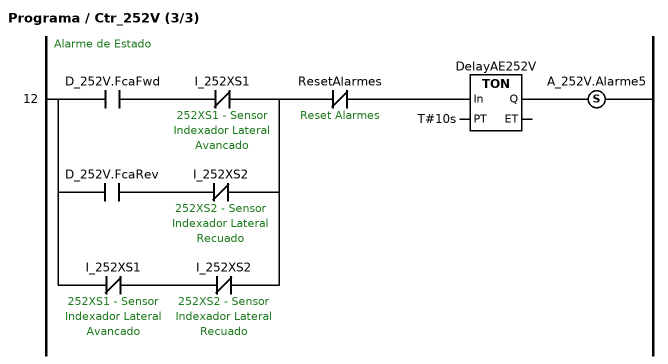
(* [picture p96: Programa / Ctr_252V, rungs 12-12] *)
(* Rung 12: Alarme de Estado *)
DelayAE252V(In := ((D_252V.FcaFwd AND NOT I_252XS1) OR (D_252V.FcaRev AND NOT I_252XS2) OR (NOT I_252XS1 AND NOT I_252XS2)) AND NOT ResetAlarmes, PT := T#10s);
IF DelayAE252V.Q THEN A_252V.Alarme5 := TRUE; END_IF;

(* Section Ctr_310M1: ladder, written here as Structured Text *)

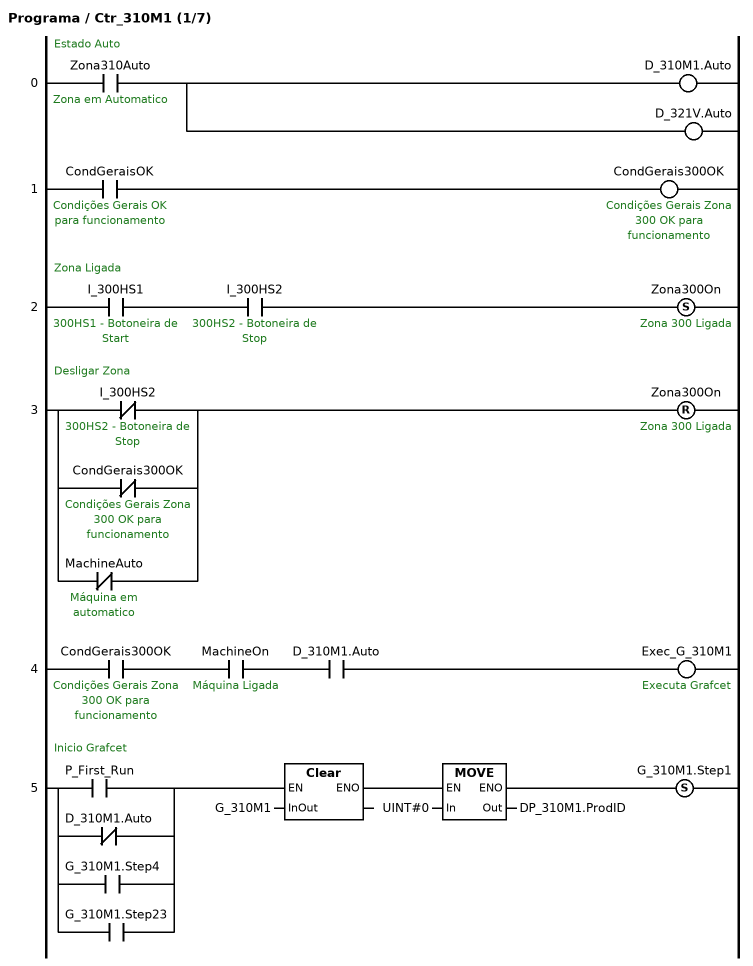
(* Rung 0: Estado Auto *)
D_310M1.Auto := Zona310Auto;
D_321V.Auto := Zona310Auto;
(* Rung 1 *)
CondGerais300OK := CondGeraisOK;
(* Rung 2: Zona Ligada *)
IF I_300HS1 AND I_300HS2 THEN Zona300On := TRUE; END_IF;
(* Rung 3: Desligar Zona *)
IF NOT I_300HS2 OR NOT CondGerais300OK OR NOT MachineAuto THEN Zona300On := FALSE; END_IF;
(* Rung 4 *)
Exec_G_310M1 := CondGerais300OK AND MachineOn AND D_310M1.Auto;
(* Rung 5: Inicio Grafcet *)
_p186 := P_First_Run OR NOT D_310M1.Auto OR G_310M1.Step4 OR G_310M1.Step23;
IF _p186 THEN
    Clear(InOut := G_310M1);
    DP_310M1.ProdID := UINT#0;
    G_310M1.Step1 := TRUE;
END_IF;

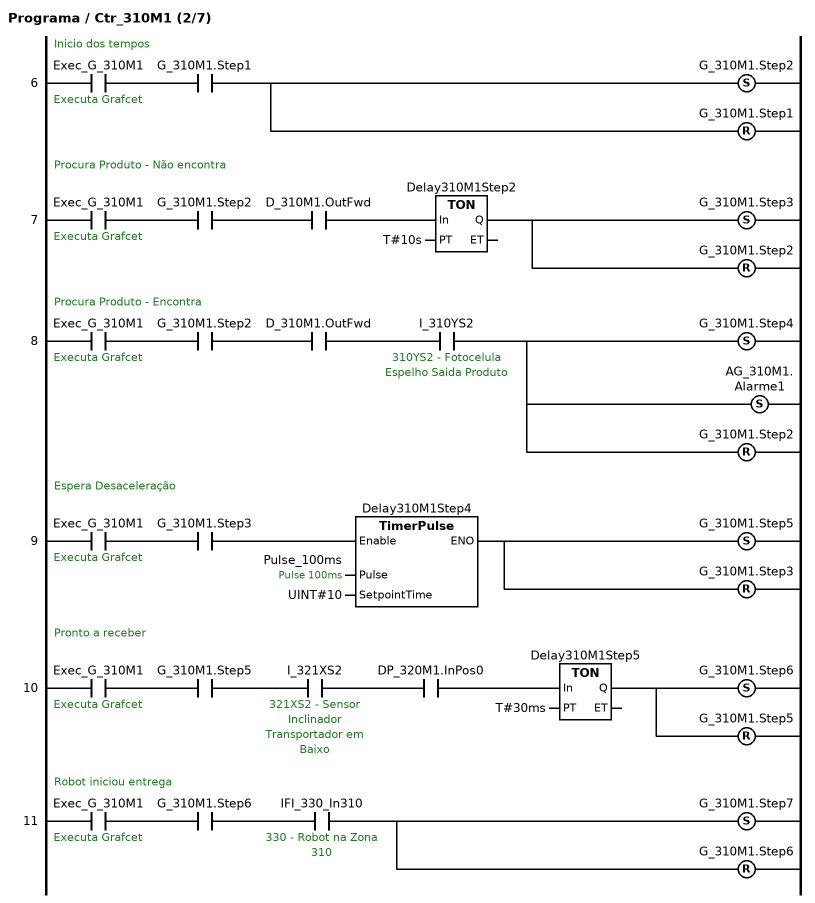
(* Rung 6: Inicio dos tempos *)
_p187 := Exec_G_310M1 AND G_310M1.Step1;
IF _p187 THEN
    G_310M1.Step2 := TRUE;
    G_310M1.Step1 := FALSE;
END_IF;
(* Rung 7: Procura Produto - Não encontra *)
Delay310M1Step2(In := Exec_G_310M1 AND G_310M1.Step2 AND D_310M1.OutFwd, PT := T#10s);
IF Delay310M1Step2.Q THEN
    G_310M1.Step3 := TRUE;
    G_310M1.Step2 := FALSE;
END_IF;
(* Rung 8: Procura Produto - Encontra *)
_p188 := Exec_G_310M1 AND G_310M1.Step2 AND D_310M1.OutFwd AND I_310YS2;
IF _p188 THEN
    G_310M1.Step4 := TRUE;
    AG_310M1.Alarme1 := TRUE;
    G_310M1.Step2 := FALSE;
END_IF;
(* Rung 9: Espera Desaceleração *)
Delay310M1Step4(Enable := Exec_G_310M1 AND G_310M1.Step3, Pulse := Pulse_100ms, SetpointTime := UINT#10);
IF Delay310M1Step4.ENO THEN
    G_310M1.Step5 := TRUE;
    G_310M1.Step3 := FALSE;
END_IF;
(* Rung 10: Pronto a receber *)
Delay310M1Step5(In := Exec_G_310M1 AND G_310M1.Step5 AND I_321XS2 AND DP_320M1.InPos0, PT := T#30ms);
IF Delay310M1Step5.Q THEN
    G_310M1.Step6 := TRUE;
    G_310M1.Step5 := FALSE;
END_IF;
(* Rung 11: Robot iniciou entrega *)
_p189 := Exec_G_310M1 AND G_310M1.Step6 AND IFI_330_In310;
IF _p189 THEN
    G_310M1.Step7 := TRUE;
    G_310M1.Step6 := FALSE;
END_IF;

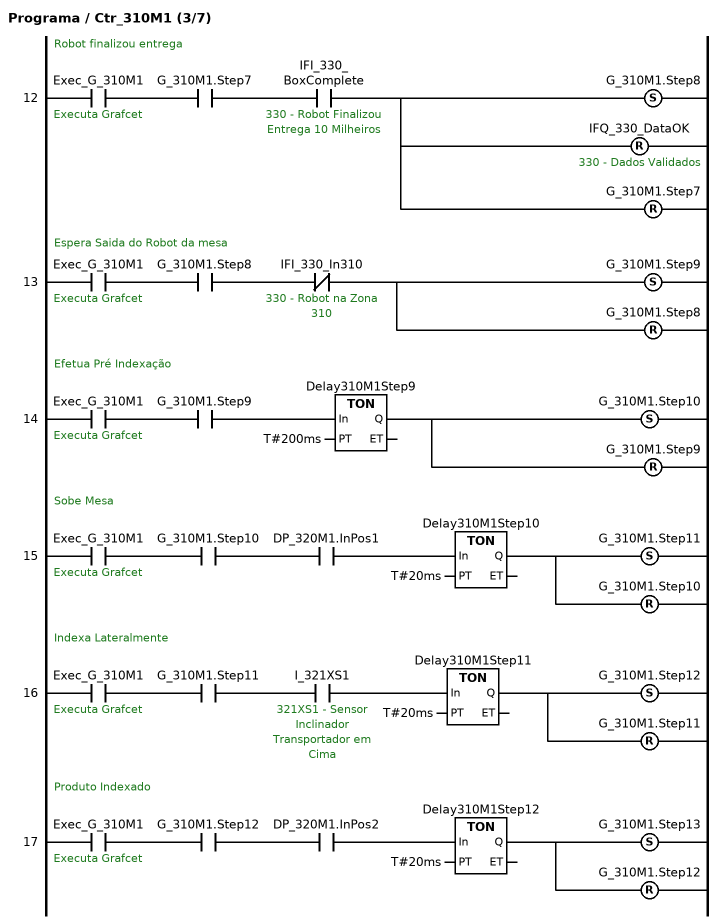
(* Rung 12: Robot finalizou entrega *)
_p190 := Exec_G_310M1 AND G_310M1.Step7 AND IFI_330_BoxComplete;
IF _p190 THEN
    G_310M1.Step8 := TRUE;
    IFQ_330_DataOK := FALSE;
    G_310M1.Step7 := FALSE;
END_IF;
(* Rung 13: Espera Saida do Robot da mesa *)
_p191 := Exec_G_310M1 AND G_310M1.Step8 AND NOT IFI_330_In310;
IF _p191 THEN
    G_310M1.Step9 := TRUE;
    G_310M1.Step8 := FALSE;
END_IF;
(* Rung 14: Efetua Pré Indexação *)
Delay310M1Step9(In := Exec_G_310M1 AND G_310M1.Step9, PT := T#200ms);
IF Delay310M1Step9.Q THEN
    G_310M1.Step10 := TRUE;
    G_310M1.Step9 := FALSE;
END_IF;
(* Rung 15: Sobe Mesa *)
Delay310M1Step10(In := Exec_G_310M1 AND G_310M1.Step10 AND DP_320M1.InPos1, PT := T#20ms);
IF Delay310M1Step10.Q THEN
    G_310M1.Step11 := TRUE;
    G_310M1.Step10 := FALSE;
END_IF;
(* Rung 16: Indexa Lateralmente *)
Delay310M1Step11(In := Exec_G_310M1 AND G_310M1.Step11 AND I_321XS1, PT := T#20ms);
IF Delay310M1Step11.Q THEN
    G_310M1.Step12 := TRUE;
    G_310M1.Step11 := FALSE;
END_IF;
(* Rung 17: Produto Indexado *)
Delay310M1Step12(In := Exec_G_310M1 AND G_310M1.Step12 AND DP_320M1.InPos2, PT := T#20ms);
IF Delay310M1Step12.Q THEN
    G_310M1.Step13 := TRUE;
    G_310M1.Step12 := FALSE;
END_IF;

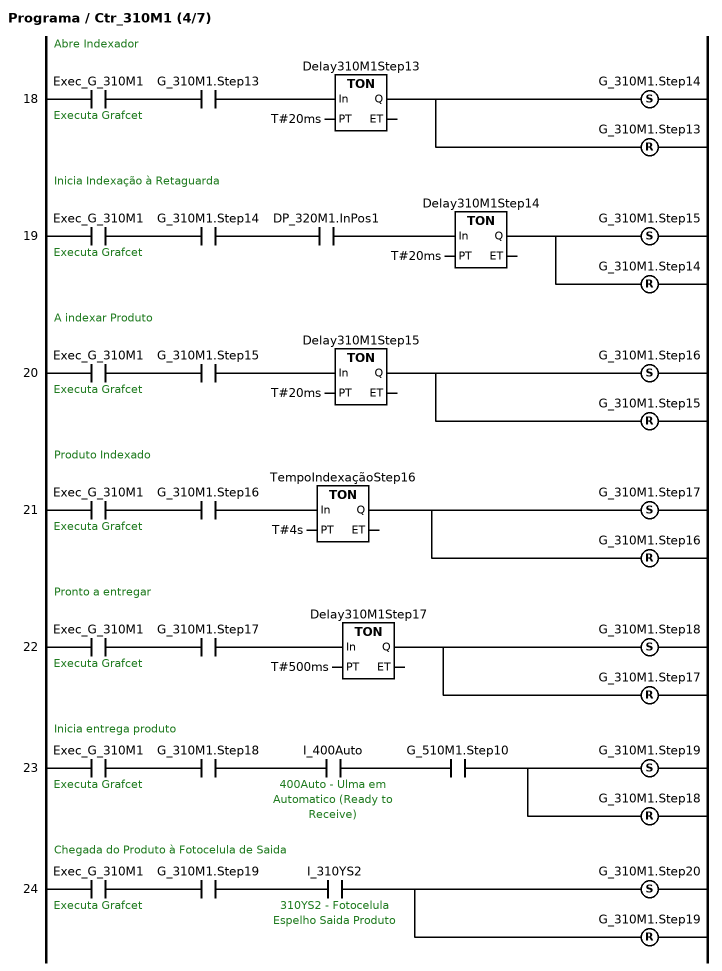
(* Rung 18: Abre Indexador *)
Delay310M1Step13(In := Exec_G_310M1 AND G_310M1.Step13, PT := T#20ms);
IF Delay310M1Step13.Q THEN
    G_310M1.Step14 := TRUE;
    G_310M1.Step13 := FALSE;
END_IF;
(* Rung 19: Inicia Indexação à Retaguarda *)
Delay310M1Step14(In := Exec_G_310M1 AND G_310M1.Step14 AND DP_320M1.InPos1, PT := T#20ms);
IF Delay310M1Step14.Q THEN
    G_310M1.Step15 := TRUE;
    G_310M1.Step14 := FALSE;
END_IF;
(* Rung 20: A indexar Produto *)
Delay310M1Step15(In := Exec_G_310M1 AND G_310M1.Step15, PT := T#20ms);
IF Delay310M1Step15.Q THEN
    G_310M1.Step16 := TRUE;
    G_310M1.Step15 := FALSE;
END_IF;
(* Rung 21: Produto Indexado *)
TempoIndexaçãoStep16(In := Exec_G_310M1 AND G_310M1.Step16, PT := T#4s);
IF TempoIndexaçãoStep16.Q THEN
    G_310M1.Step17 := TRUE;
    G_310M1.Step16 := FALSE;
END_IF;
(* Rung 22: Pronto a entregar *)
Delay310M1Step17(In := Exec_G_310M1 AND G_310M1.Step17, PT := T#500ms);
IF Delay310M1Step17.Q THEN
    G_310M1.Step18 := TRUE;
    G_310M1.Step17 := FALSE;
END_IF;
(* Rung 23: Inicia entrega produto *)
_p192 := Exec_G_310M1 AND G_310M1.Step18 AND I_400Auto AND G_510M1.Step10;
IF _p192 THEN
    G_310M1.Step19 := TRUE;
    G_310M1.Step18 := FALSE;
END_IF;
(* Rung 24: Chegada do Produto à Fotocelula de Saida *)
_p193 := Exec_G_310M1 AND G_310M1.Step19 AND I_310YS2;
IF _p193 THEN
    G_310M1.Step20 := TRUE;
    G_310M1.Step19 := FALSE;
END_IF;

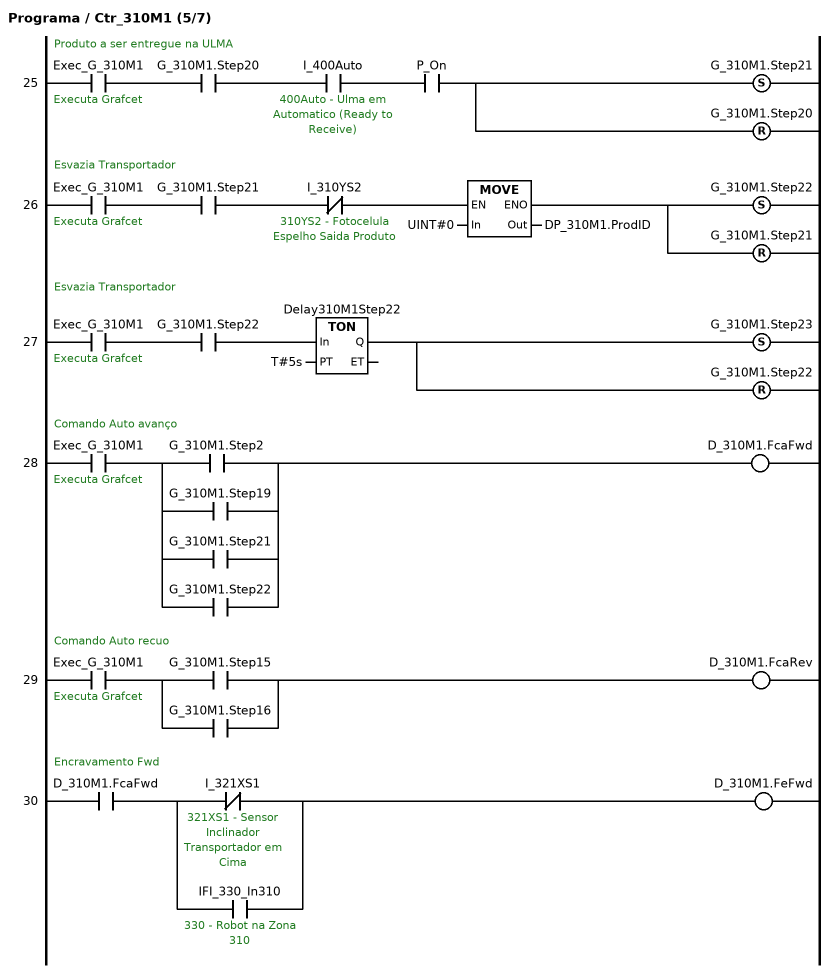
(* Rung 25: Produto a ser entregue na ULMA *)
_p194 := Exec_G_310M1 AND G_310M1.Step20 AND I_400Auto AND P_On;
IF _p194 THEN
    G_310M1.Step21 := TRUE;
    G_310M1.Step20 := FALSE;
END_IF;
(* Rung 26: Esvazia Transportador *)
IF Exec_G_310M1 AND G_310M1.Step21 AND NOT I_310YS2 THEN DP_310M1.ProdID := UINT#0; END_IF;
_p195 := Exec_G_310M1 AND G_310M1.Step21 AND NOT I_310YS2;
IF _p195 THEN
    G_310M1.Step22 := TRUE;
    G_310M1.Step21 := FALSE;
END_IF;
(* Rung 27: Esvazia Transportador *)
Delay310M1Step22(In := Exec_G_310M1 AND G_310M1.Step22, PT := T#5s);
IF Delay310M1Step22.Q THEN
    G_310M1.Step23 := TRUE;
    G_310M1.Step22 := FALSE;
END_IF;
(* Rung 28: Comando Auto avanço *)
D_310M1.FcaFwd := Exec_G_310M1 AND (G_310M1.Step2 OR G_310M1.Step19 OR G_310M1.Step21 OR G_310M1.Step22);
(* Rung 29: Comando Auto recuo *)
D_310M1.FcaRev := Exec_G_310M1 AND (G_310M1.Step15 OR G_310M1.Step16);
(* Rung 30: Encravamento Fwd *)
D_310M1.FeFwd := D_310M1.FcaFwd AND (NOT I_321XS1 OR IFI_330_In310);

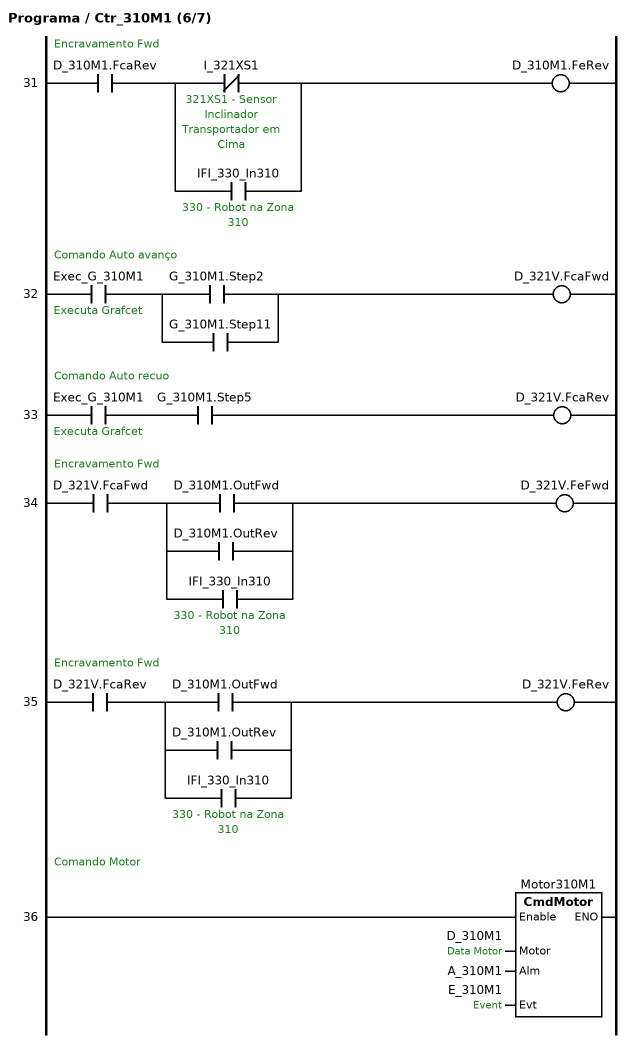
(* Rung 31: Encravamento Fwd *)
D_310M1.FeRev := D_310M1.FcaRev AND (NOT I_321XS1 OR IFI_330_In310);
(* Rung 32: Comando Auto avanço *)
D_321V.FcaFwd := Exec_G_310M1 AND (G_310M1.Step2 OR G_310M1.Step11);
(* Rung 33: Comando Auto recuo *)
D_321V.FcaRev := Exec_G_310M1 AND G_310M1.Step5;
(* Rung 34: Encravamento Fwd *)
D_321V.FeFwd := D_321V.FcaFwd AND (D_310M1.OutFwd OR D_310M1.OutRev OR IFI_330_In310);
(* Rung 35: Encravamento Fwd *)
D_321V.FeRev := D_321V.FcaRev AND (D_310M1.OutFwd OR D_310M1.OutRev OR IFI_330_In310);
(* Rung 36: Comando Motor *)
Motor310M1(Enable := TRUE, Motor := D_310M1, Alm := A_310M1, Evt := E_310M1);

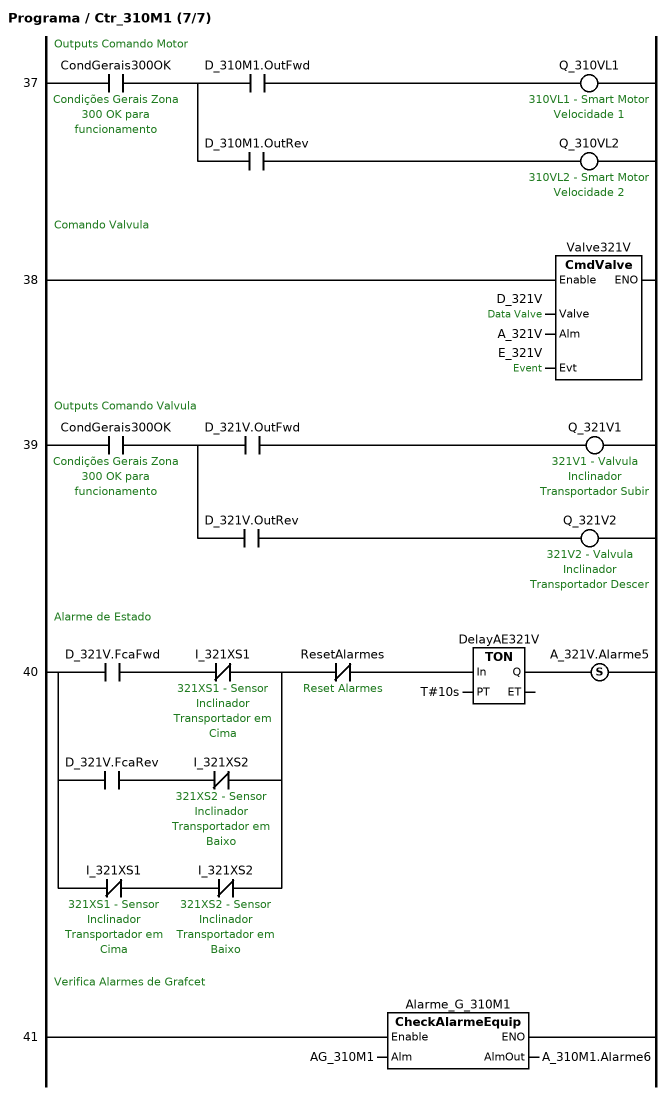
(* Rung 37: Outputs Comando Motor *)
Q_310VL1 := CondGerais300OK AND D_310M1.OutFwd;
Q_310VL2 := CondGerais300OK AND D_310M1.OutRev;
(* Rung 38: Comando Valvula *)
Valve321V(Enable := TRUE, Valve := D_321V, Alm := A_321V, Evt := E_321V);
(* Rung 39: Outputs Comando Valvula *)
Q_321V1 := CondGerais300OK AND D_321V.OutFwd;
Q_321V2 := CondGerais300OK AND D_321V.OutRev;
(* Rung 40: Alarme de Estado *)
DelayAE321V(In := ((D_321V.FcaFwd AND NOT I_321XS1) OR (D_321V.FcaRev AND NOT I_321XS2) OR (NOT I_321XS1 AND NOT I_321XS2)) AND NOT ResetAlarmes, PT := T#10s);
IF DelayAE321V.Q THEN A_321V.Alarme5 := TRUE; END_IF;
(* Rung 41: Verifica Alarmes de Grafcet *)
Alarme_G_310M1(Enable := TRUE, Alm := AG_310M1, AlmOut => A_310M1.Alarme6);

(* Section Ctr_320M1_Servo: ladder, written here as Structured Text *)

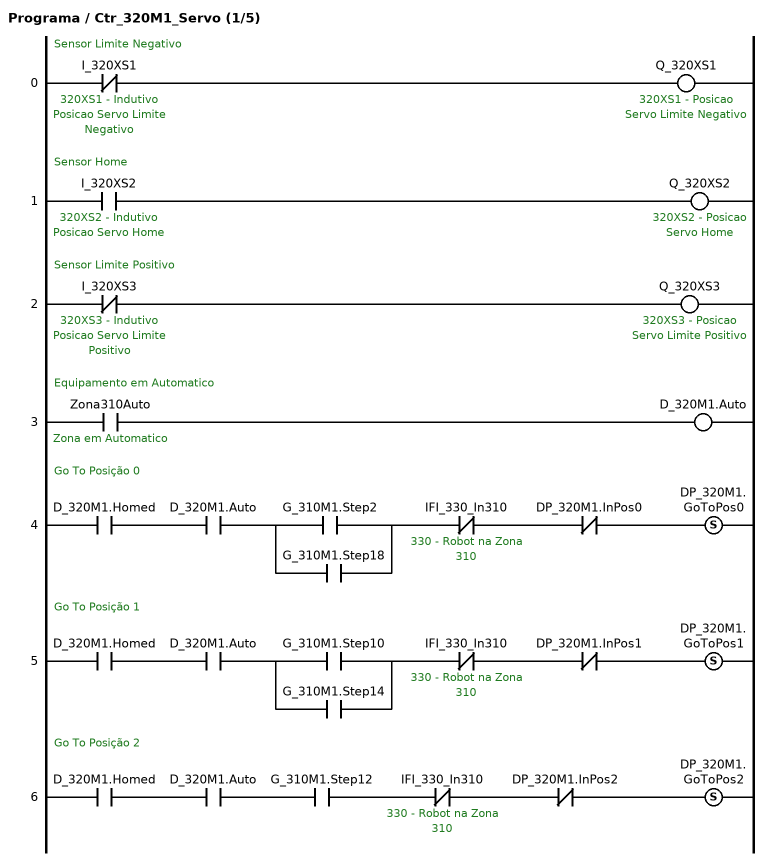
(* Rung 0: Sensor Limite Negativo *)
Q_320XS1 := NOT I_320XS1;
(* Rung 1: Sensor Home *)
Q_320XS2 := I_320XS2;
(* Rung 2: Sensor Limite Positivo *)
Q_320XS3 := NOT I_320XS3;
(* Rung 3: Equipamento em Automatico *)
D_320M1.Auto := Zona310Auto;
(* Rung 4: Go To Posição 0 *)
IF D_320M1.Homed AND D_320M1.Auto AND (G_310M1.Step2 OR G_310M1.Step18) AND NOT IFI_330_In310 AND NOT DP_320M1.InPos0 THEN
    DP_320M1.GoToPos0 := TRUE;
END_IF;
(* Rung 5: Go To Posição 1 *)
IF D_320M1.Homed AND D_320M1.Auto AND (G_310M1.Step10 OR G_310M1.Step14) AND NOT IFI_330_In310 AND NOT DP_320M1.InPos1 THEN
    DP_320M1.GoToPos1 := TRUE;
END_IF;
(* Rung 6: Go To Posição 2 *)
IF D_320M1.Homed AND D_320M1.Auto AND G_310M1.Step12 AND NOT IFI_330_In310 AND NOT DP_320M1.InPos2 THEN
    DP_320M1.GoToPos2 := TRUE;
END_IF;

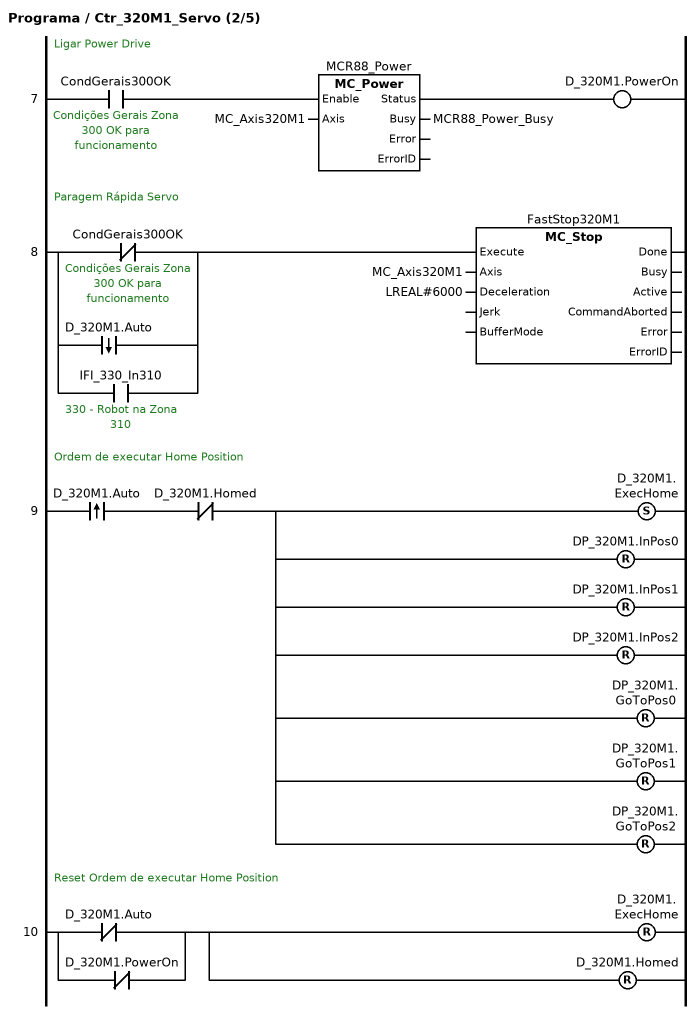
(* Rung 7: Ligar Power Drive *)
MCR88_Power(Enable := CondGerais300OK, Axis := MC_Axis320M1, Busy => MCR88_Power_Busy);
D_320M1.PowerOn := MCR88_Power.Status;
(* Rung 8: Paragem Rápida Servo *)
_e196(CLK := D_320M1.Auto);
FastStop320M1(Execute := NOT CondGerais300OK OR _e196.Q OR IFI_330_In310, Axis := MC_Axis320M1, Deceleration := LREAL#6000);
(* Rung 9: Ordem de executar Home Position *)
_e197(CLK := D_320M1.Auto);
_p198 := _e197.Q AND NOT D_320M1.Homed;
IF _p198 THEN
    D_320M1.ExecHome := TRUE;
    DP_320M1.InPos0 := FALSE;
    DP_320M1.InPos1 := FALSE;
    DP_320M1.InPos2 := FALSE;
    DP_320M1.GoToPos0 := FALSE;
    DP_320M1.GoToPos1 := FALSE;
    DP_320M1.GoToPos2 := FALSE;
END_IF;
(* Rung 10: Reset Ordem de executar Home Position *)
_p199 := NOT D_320M1.Auto OR NOT D_320M1.PowerOn;
IF _p199 THEN
    D_320M1.ExecHome := FALSE;
    D_320M1.Homed := FALSE;
END_IF;

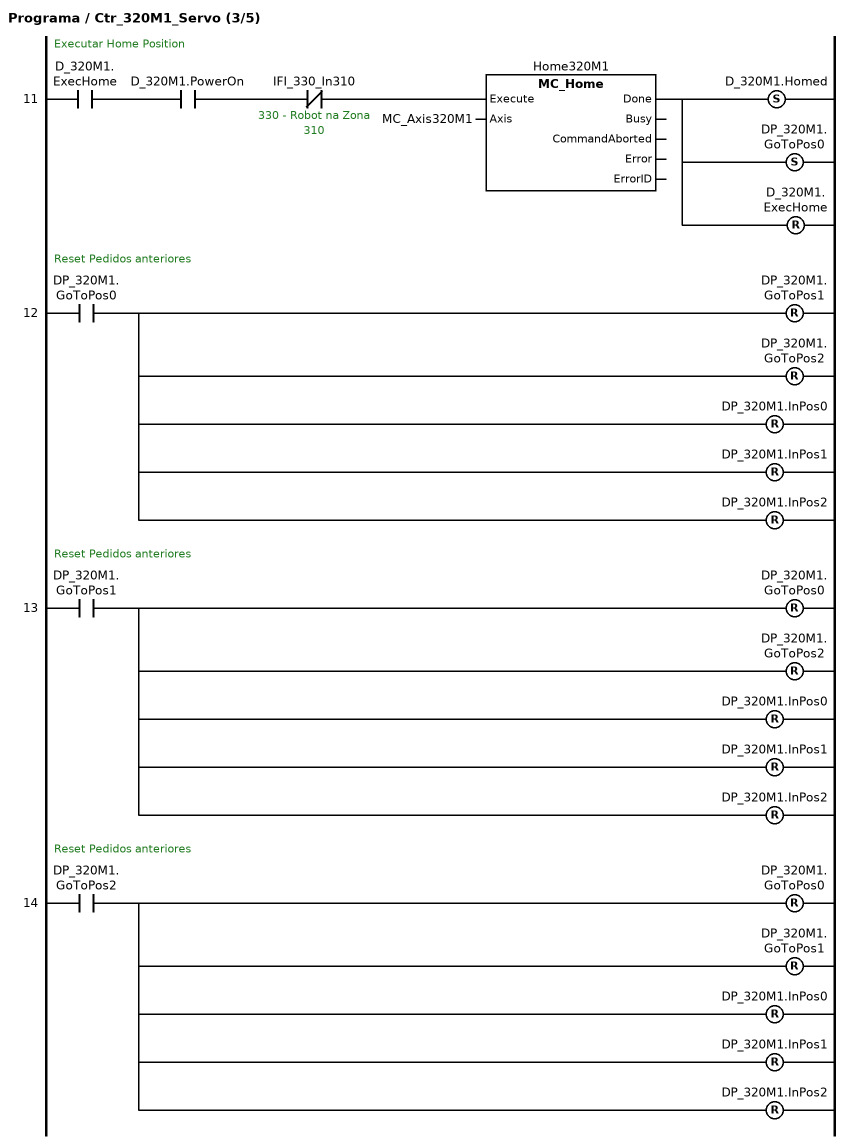
(* Rung 11: Executar Home Position *)
Home320M1(Execute := D_320M1.ExecHome AND D_320M1.PowerOn AND NOT IFI_330_In310, Axis := MC_Axis320M1);
IF Home320M1.Done THEN
    D_320M1.Homed := TRUE;
    DP_320M1.GoToPos0 := TRUE;
    D_320M1.ExecHome := FALSE;
END_IF;
(* Rung 12: Reset Pedidos anteriores *)
_p200 := DP_320M1.GoToPos0;
IF _p200 THEN
    DP_320M1.GoToPos1 := FALSE;
    DP_320M1.GoToPos2 := FALSE;
    DP_320M1.InPos0 := FALSE;
    DP_320M1.InPos1 := FALSE;
    DP_320M1.InPos2 := FALSE;
END_IF;
(* Rung 13: Reset Pedidos anteriores *)
_p201 := DP_320M1.GoToPos1;
IF _p201 THEN
    DP_320M1.GoToPos0 := FALSE;
    DP_320M1.GoToPos2 := FALSE;
    DP_320M1.InPos0 := FALSE;
    DP_320M1.InPos1 := FALSE;
    DP_320M1.InPos2 := FALSE;
END_IF;
(* Rung 14: Reset Pedidos anteriores *)
_p202 := DP_320M1.GoToPos2;
IF _p202 THEN
    DP_320M1.GoToPos0 := FALSE;
    DP_320M1.GoToPos1 := FALSE;
    DP_320M1.InPos0 := FALSE;
    DP_320M1.InPos1 := FALSE;
    DP_320M1.InPos2 := FALSE;
END_IF;

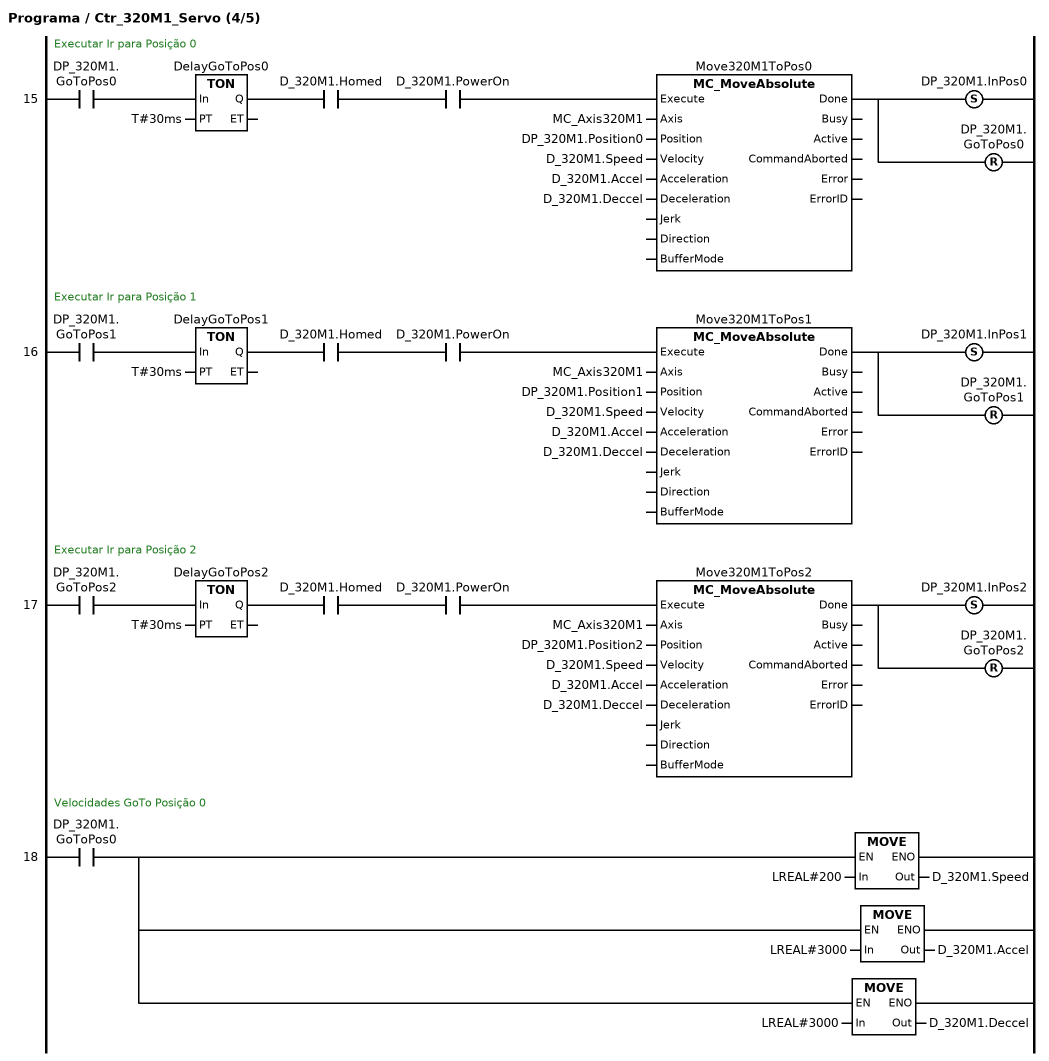
(* Rung 15: Executar Ir para Posição 0 *)
DelayGoToPos0(In := DP_320M1.GoToPos0, PT := T#30ms);
Move320M1ToPos0(Execute := DelayGoToPos0.Q AND D_320M1.Homed AND D_320M1.PowerOn, Axis := MC_Axis320M1, Position := DP_320M1.Position0, Velocity := D_320M1.Speed, Acceleration := D_320M1.Accel, Deceleration := D_320M1.Deccel);
IF Move320M1ToPos0.Done THEN
    DP_320M1.InPos0 := TRUE;
    DP_320M1.GoToPos0 := FALSE;
END_IF;
(* Rung 16: Executar Ir para Posição 1 *)
DelayGoToPos1(In := DP_320M1.GoToPos1, PT := T#30ms);
Move320M1ToPos1(Execute := DelayGoToPos1.Q AND D_320M1.Homed AND D_320M1.PowerOn, Axis := MC_Axis320M1, Position := DP_320M1.Position1, Velocity := D_320M1.Speed, Acceleration := D_320M1.Accel, Deceleration := D_320M1.Deccel);
IF Move320M1ToPos1.Done THEN
    DP_320M1.InPos1 := TRUE;
    DP_320M1.GoToPos1 := FALSE;
END_IF;
(* Rung 17: Executar Ir para Posição 2 *)
DelayGoToPos2(In := DP_320M1.GoToPos2, PT := T#30ms);
Move320M1ToPos2(Execute := DelayGoToPos2.Q AND D_320M1.Homed AND D_320M1.PowerOn, Axis := MC_Axis320M1, Position := DP_320M1.Position2, Velocity := D_320M1.Speed, Acceleration := D_320M1.Accel, Deceleration := D_320M1.Deccel);
IF Move320M1ToPos2.Done THEN
    DP_320M1.InPos2 := TRUE;
    DP_320M1.GoToPos2 := FALSE;
END_IF;
(* Rung 18: Velocidades GoTo Posição 0 *)
IF DP_320M1.GoToPos0 THEN
    D_320M1.Speed := LREAL#200;
    D_320M1.Accel := LREAL#3000;
    D_320M1.Deccel := LREAL#3000;
END_IF;

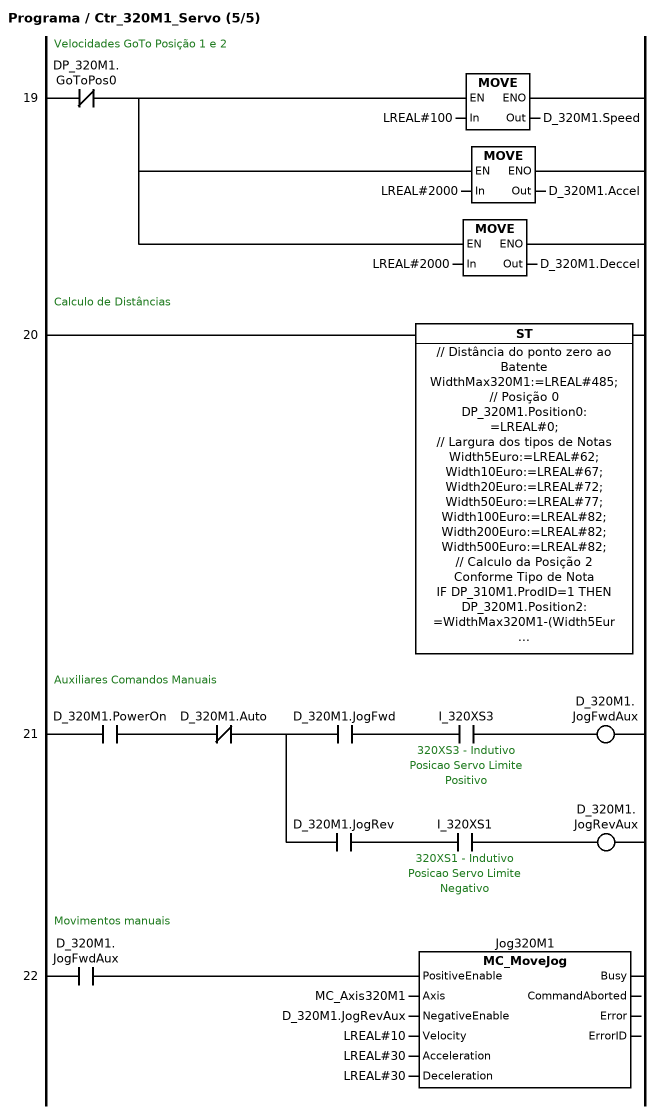
(* Rung 19: Velocidades GoTo Posição 1 e 2 *)
IF NOT DP_320M1.GoToPos0 THEN
    D_320M1.Speed := LREAL#100;
    D_320M1.Accel := LREAL#2000;
    D_320M1.Deccel := LREAL#2000;
END_IF;
(* Rung 20: Calculo de Distâncias *)
// Distância do ponto zero ao Batente

WidthMax320M1:=LREAL#485;

// Posição 0

DP_320M1.Position0:=LREAL#0;

// Largura dos tipos de Notas

Width5Euro:=LREAL#62;
Width10Euro:=LREAL#67;
Width20Euro:=LREAL#72;
Width50Euro:=LREAL#77;
Width100Euro:=LREAL#82;
Width200Euro:=LREAL#82;
Width500Euro:=LREAL#82;

// Calculo da Posição 2 Conforme Tipo de Nota

IF DP_310M1.ProdID=1 THEN DP_320M1.Position2:=WidthMax320M1-(Width5Euro*5); END_IF;
IF DP_310M1.ProdID=2 THEN DP_320M1.Position2:=WidthMax320M1-(Width10Euro*5); END_IF;
IF DP_310M1.ProdID=3 THEN DP_320M1.Position2:=WidthMax320M1-(Width20Euro*5); END_IF;	
IF DP_310M1.ProdID=4 THEN DP_320M1.Position2:=WidthMax320M1-(Width50Euro*5); END_IF;	
IF DP_310M1.ProdID=5 THEN DP_320M1.Position2:=WidthMax320M1-(Width100Euro*5); END_IF;
IF DP_310M1.ProdID=6 THEN DP_320M1.Position2:=WidthMax320M1-(Width200Euro*5); END_IF;
IF DP_310M1.ProdID=7 THEN DP_320M1.Position2:=WidthMax320M1-(Width500Euro*5); END_IF;
IF DP_310M1.ProdID<1 OR DP_310M1.ProdID>7 THEN DP_320M1.Position2:=WidthMax320M1-(Width500Euro*5); END_IF;
	
// Calculo da Posição 1 relativa a Posição 2

DP_320M1.Position1:=DP_320M1.Position2-LREAL#20;
(* Rung 21: Auxiliares Comandos Manuais *)
_p203 := D_320M1.PowerOn AND NOT D_320M1.Auto;
D_320M1.JogFwdAux := D_320M1.PowerOn AND NOT D_320M1.Auto AND D_320M1.JogFwd AND I_320XS3;
D_320M1.JogRevAux := _p203 AND D_320M1.JogRev AND I_320XS1;
(* Rung 22: Movimentos manuais *)
Jog320M1(PositiveEnable := D_320M1.JogFwdAux, Axis := MC_Axis320M1, NegativeEnable := D_320M1.JogRevAux, Velocity := LREAL#10, Acceleration := LREAL#30, Deceleration := LREAL#30);

(* Section InterfaceRobot: ladder, written here as Structured Text *)

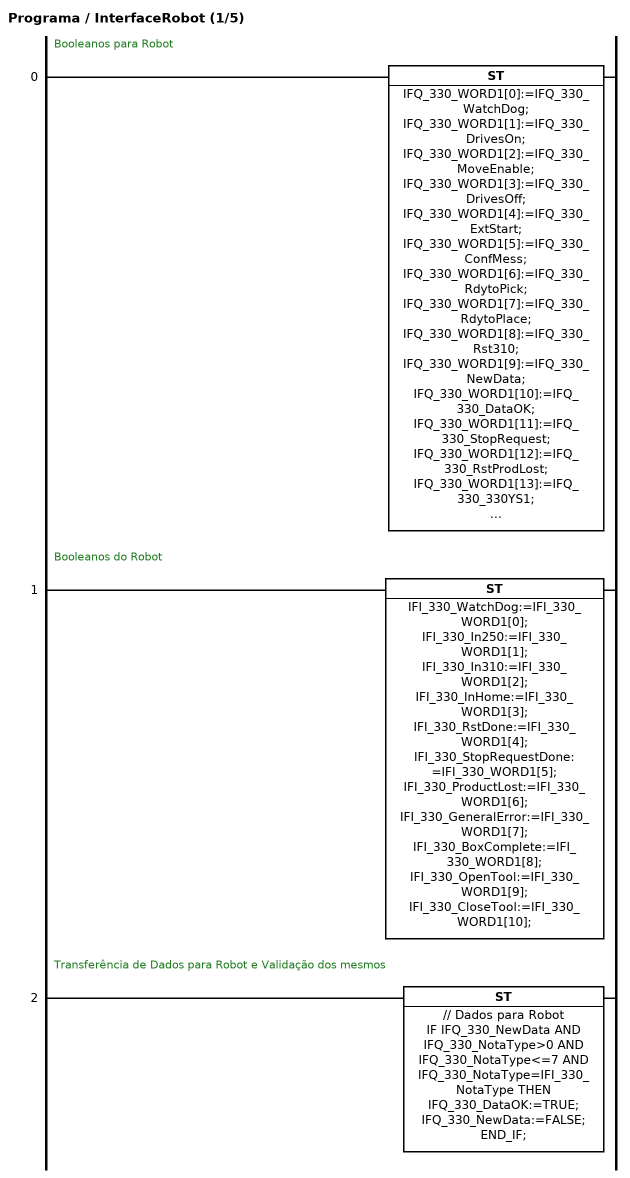
(* Rung 0: Booleanos para Robot *)
IFQ_330_WORD1[0]:=IFQ_330_WatchDog;
IFQ_330_WORD1[1]:=IFQ_330_DrivesOn;
IFQ_330_WORD1[2]:=IFQ_330_MoveEnable;
IFQ_330_WORD1[3]:=IFQ_330_DrivesOff;
IFQ_330_WORD1[4]:=IFQ_330_ExtStart;
IFQ_330_WORD1[5]:=IFQ_330_ConfMess;
IFQ_330_WORD1[6]:=IFQ_330_RdytoPick;
IFQ_330_WORD1[7]:=IFQ_330_RdytoPlace;
IFQ_330_WORD1[8]:=IFQ_330_Rst310;
IFQ_330_WORD1[9]:=IFQ_330_NewData;
IFQ_330_WORD1[10]:=IFQ_330_DataOK;
IFQ_330_WORD1[11]:=IFQ_330_StopRequest;
IFQ_330_WORD1[12]:=IFQ_330_RstProdLost;
IFQ_330_WORD1[13]:=IFQ_330_330YS1;
IFQ_330_WORD1[14]:=IFQ_330_330YS2;
IFQ_330_WORD1[15]:=IFQ_330_330XS1;
(* Rung 1: Booleanos do Robot *)
IFI_330_WatchDog:=IFI_330_WORD1[0];
IFI_330_In250:=IFI_330_WORD1[1];
IFI_330_In310:=IFI_330_WORD1[2];
IFI_330_InHome:=IFI_330_WORD1[3];
IFI_330_RstDone:=IFI_330_WORD1[4];
IFI_330_StopRequestDone:=IFI_330_WORD1[5];
IFI_330_ProductLost:=IFI_330_WORD1[6];
IFI_330_GeneralError:=IFI_330_WORD1[7];
IFI_330_BoxComplete:=IFI_330_WORD1[8];
IFI_330_OpenTool:=IFI_330_WORD1[9];
IFI_330_CloseTool:=IFI_330_WORD1[10];
(* Rung 2: Transferência de Dados para Robot e Validação dos mesmos *)
// Dados para Robot

IF IFQ_330_NewData AND IFQ_330_NotaType>0 AND IFQ_330_NotaType<=7 AND
	IFQ_330_NotaType=IFI_330_NotaType THEN
	IFQ_330_DataOK:=TRUE;
	IFQ_330_NewData:=FALSE;
END_IF;

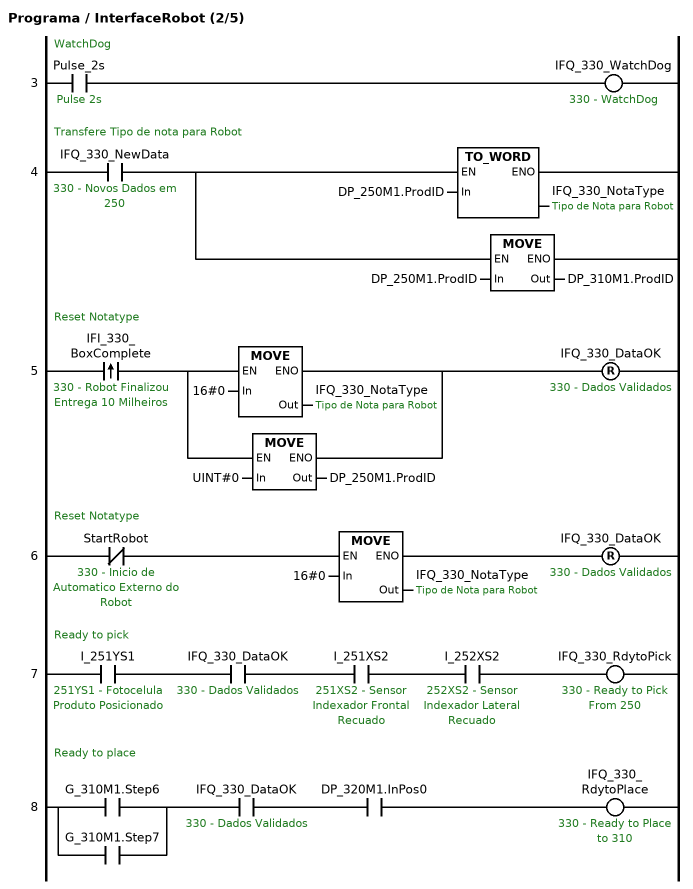
(* Rung 3: WatchDog *)
IFQ_330_WatchDog := Pulse_2s;
(* Rung 4: Transfere Tipo de nota para Robot *)
IF IFQ_330_NewData THEN
    IFQ_330_NotaType := TO_WORD(In := DP_250M1.ProdID);
    DP_310M1.ProdID := DP_250M1.ProdID;
END_IF;
(* Rung 5: Reset Notatype *)
_e204(CLK := IFI_330_BoxComplete);
IF _e204.Q THEN
    IFQ_330_NotaType := 16#0;
    DP_250M1.ProdID := UINT#0;
    IFQ_330_DataOK := FALSE;
END_IF;
(* Rung 6: Reset Notatype *)
IF NOT StartRobot THEN
    IFQ_330_NotaType := 16#0;
    IFQ_330_DataOK := FALSE;
END_IF;
(* Rung 7: Ready to pick *)
IFQ_330_RdytoPick := I_251YS1 AND IFQ_330_DataOK AND I_251XS2 AND I_252XS2;
(* Rung 8: Ready to place *)
IFQ_330_RdytoPlace := (G_310M1.Step6 OR G_310M1.Step7) AND IFQ_330_DataOK AND DP_320M1.InPos0;

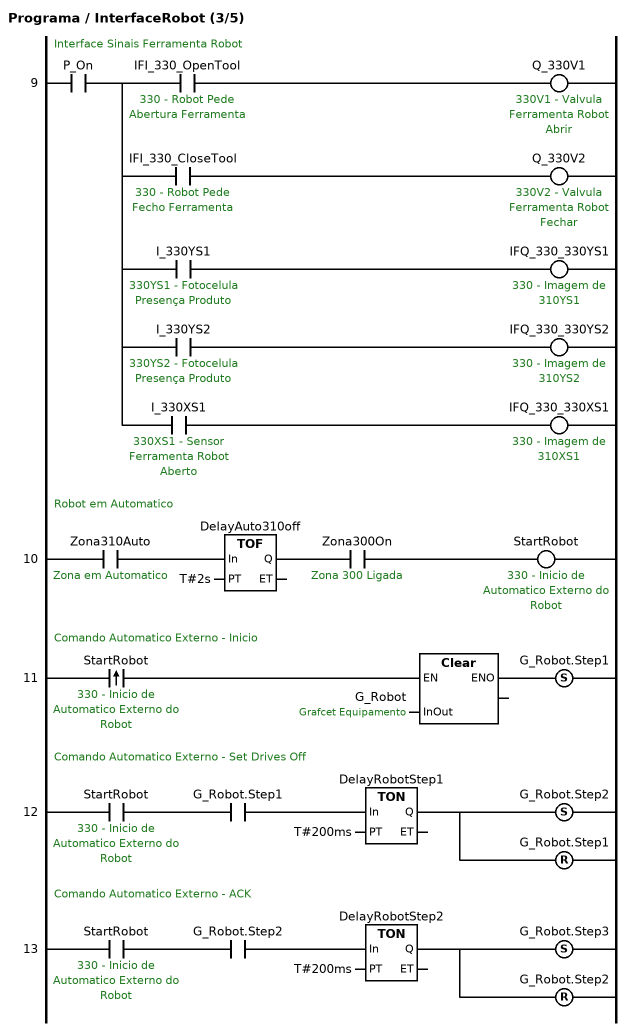
(* Rung 9: Interface Sinais Ferramenta Robot *)
Q_330V1 := P_On AND IFI_330_OpenTool;
Q_330V2 := P_On AND IFI_330_CloseTool;
IFQ_330_330YS1 := P_On AND I_330YS1;
IFQ_330_330YS2 := P_On AND I_330YS2;
IFQ_330_330XS1 := P_On AND I_330XS1;
(* Rung 10: Robot em Automatico *)
DelayAuto310off(In := Zona310Auto, PT := T#2s);
StartRobot := DelayAuto310off.Q AND Zona300On;
(* Rung 11: Comando Automatico Externo - Inicio *)
_e205(CLK := StartRobot);
IF _e205.Q THEN
    Clear(InOut := G_Robot);
    G_Robot.Step1 := TRUE;
END_IF;
(* Rung 12: Comando Automatico Externo - Set Drives Off *)
DelayRobotStep1(In := StartRobot AND G_Robot.Step1, PT := T#200ms);
IF DelayRobotStep1.Q THEN
    G_Robot.Step2 := TRUE;
    G_Robot.Step1 := FALSE;
END_IF;
(* Rung 13: Comando Automatico Externo - ACK *)
DelayRobotStep2(In := StartRobot AND G_Robot.Step2, PT := T#200ms);
IF DelayRobotStep2.Q THEN
    G_Robot.Step3 := TRUE;
    G_Robot.Step2 := FALSE;
END_IF;

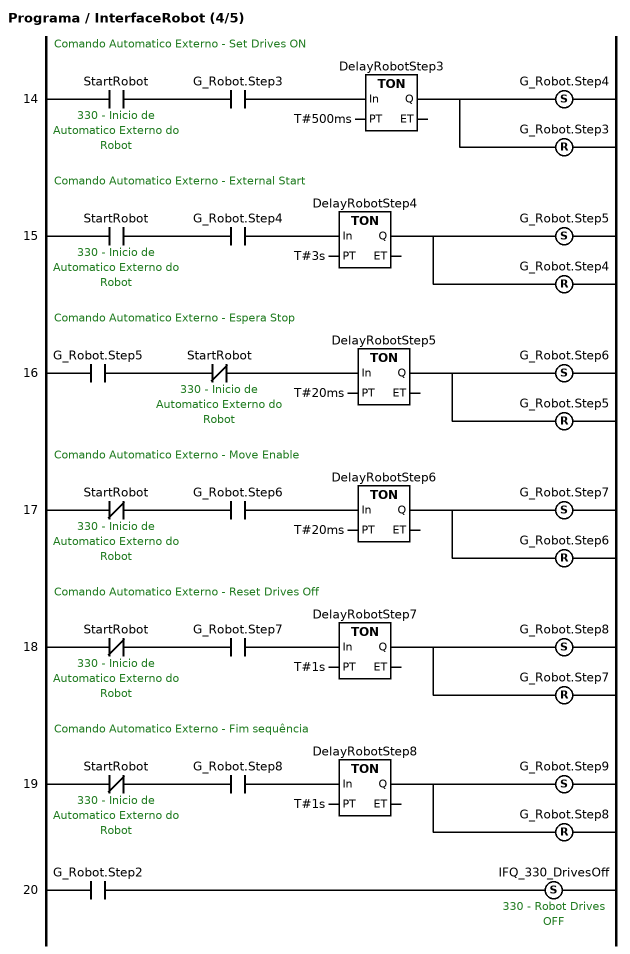
(* Rung 14: Comando Automatico Externo - Set Drives ON *)
DelayRobotStep3(In := StartRobot AND G_Robot.Step3, PT := T#500ms);
IF DelayRobotStep3.Q THEN
    G_Robot.Step4 := TRUE;
    G_Robot.Step3 := FALSE;
END_IF;
(* Rung 15: Comando Automatico Externo - External Start *)
DelayRobotStep4(In := StartRobot AND G_Robot.Step4, PT := T#3s);
IF DelayRobotStep4.Q THEN
    G_Robot.Step5 := TRUE;
    G_Robot.Step4 := FALSE;
END_IF;
(* Rung 16: Comando Automatico Externo - Espera Stop *)
DelayRobotStep5(In := G_Robot.Step5 AND NOT StartRobot, PT := T#20ms);
IF DelayRobotStep5.Q THEN
    G_Robot.Step6 := TRUE;
    G_Robot.Step5 := FALSE;
END_IF;
(* Rung 17: Comando Automatico Externo - Move Enable *)
DelayRobotStep6(In := NOT StartRobot AND G_Robot.Step6, PT := T#20ms);
IF DelayRobotStep6.Q THEN
    G_Robot.Step7 := TRUE;
    G_Robot.Step6 := FALSE;
END_IF;
(* Rung 18: Comando Automatico Externo - Reset Drives Off *)
DelayRobotStep7(In := NOT StartRobot AND G_Robot.Step7, PT := T#1s);
IF DelayRobotStep7.Q THEN
    G_Robot.Step8 := TRUE;
    G_Robot.Step7 := FALSE;
END_IF;
(* Rung 19: Comando Automatico Externo - Fim sequência *)
DelayRobotStep8(In := NOT StartRobot AND G_Robot.Step8, PT := T#1s);
IF DelayRobotStep8.Q THEN
    G_Robot.Step9 := TRUE;
    G_Robot.Step8 := FALSE;
END_IF;
(* Rung 20 *)
IF G_Robot.Step2 THEN IFQ_330_DrivesOff := TRUE; END_IF;

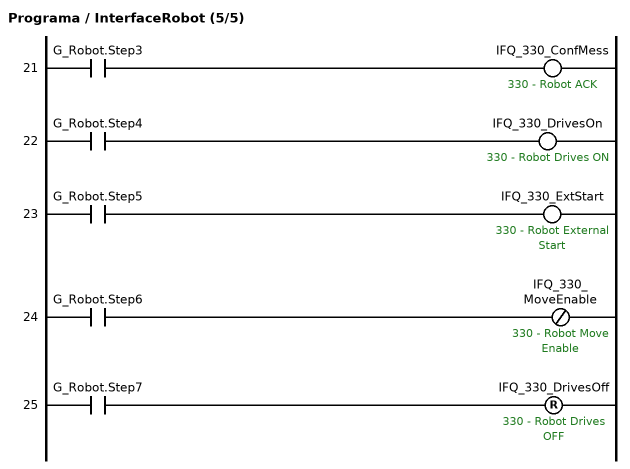
(* Rung 21 *)
IFQ_330_ConfMess := G_Robot.Step3;
(* Rung 22 *)
IFQ_330_DrivesOn := G_Robot.Step4;
(* Rung 23 *)
IFQ_330_ExtStart := G_Robot.Step5;
(* Rung 24 *)
IFQ_330_MoveEnable := NOT G_Robot.Step6;
(* Rung 25 *)
IF G_Robot.Step7 THEN IFQ_330_DrivesOff := FALSE; END_IF;

(* Section InterfaceHMI: ladder, written here as Structured Text *)

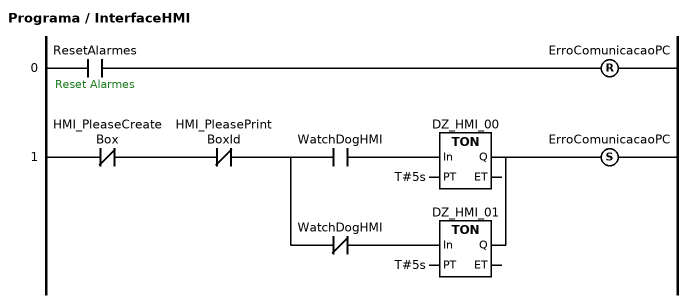
(* Rung 0 *)
IF ResetAlarmes THEN ErroComunicacaoPC := FALSE; END_IF;
(* Rung 1 *)
_p206 := NOT HMI_PleaseCreateBox AND NOT HMI_PleasePrintBoxId;
DZ_HMI_00(In := _p206 AND WatchDogHMI, PT := T#5s);
DZ_HMI_01(In := _p206 AND NOT WatchDogHMI, PT := T#5s);
IF DZ_HMI_00.Q OR DZ_HMI_01.Q THEN ErroComunicacaoPC := TRUE; END_IF;

(* Section Ctr_510M1: ladder, written here as Structured Text *)

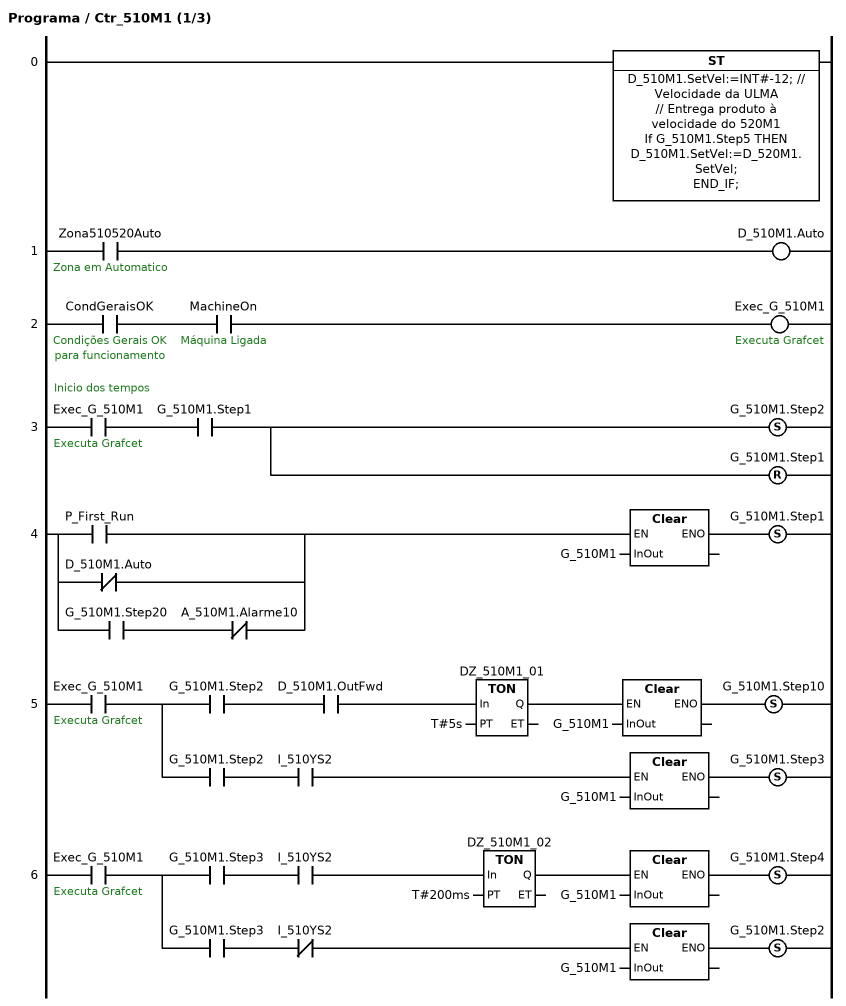
(* Rung 0 *)
D_510M1.SetVel:=INT#-12; // Velocidade da ULMA
// Entrega produto à velocidade do 520M1
If G_510M1.Step5 THEN
	D_510M1.SetVel:=D_520M1.SetVel;
END_IF;
	
(* Rung 1 *)
D_510M1.Auto := Zona510520Auto;
(* Rung 2 *)
Exec_G_510M1 := CondGeraisOK AND MachineOn;
(* Rung 3: Inicio dos tempos *)
_p207 := Exec_G_510M1 AND G_510M1.Step1;
IF _p207 THEN
    G_510M1.Step2 := TRUE;
    G_510M1.Step1 := FALSE;
END_IF;
(* Rung 4 *)
_p208 := P_First_Run OR NOT D_510M1.Auto OR (G_510M1.Step20 AND NOT A_510M1.Alarme10);
IF _p208 THEN
    Clear(InOut := G_510M1);
    G_510M1.Step1 := TRUE;
END_IF;
(* Rung 5 *)
DZ_510M1_01(In := Exec_G_510M1 AND G_510M1.Step2 AND D_510M1.OutFwd, PT := T#5s);
IF DZ_510M1_01.Q THEN
    Clear(InOut := G_510M1);
    G_510M1.Step10 := TRUE;
END_IF;
_p209 := Exec_G_510M1 AND G_510M1.Step2 AND I_510YS2;
IF _p209 THEN
    Clear(InOut := G_510M1);
    G_510M1.Step3 := TRUE;
END_IF;
(* Rung 6 *)
DZ_510M1_02(In := Exec_G_510M1 AND G_510M1.Step3 AND I_510YS2, PT := T#200ms);
IF DZ_510M1_02.Q THEN
    Clear(InOut := G_510M1);
    G_510M1.Step4 := TRUE;
END_IF;
_p210 := Exec_G_510M1 AND G_510M1.Step3 AND NOT I_510YS2;
IF _p210 THEN
    Clear(InOut := G_510M1);
    G_510M1.Step2 := TRUE;
END_IF;

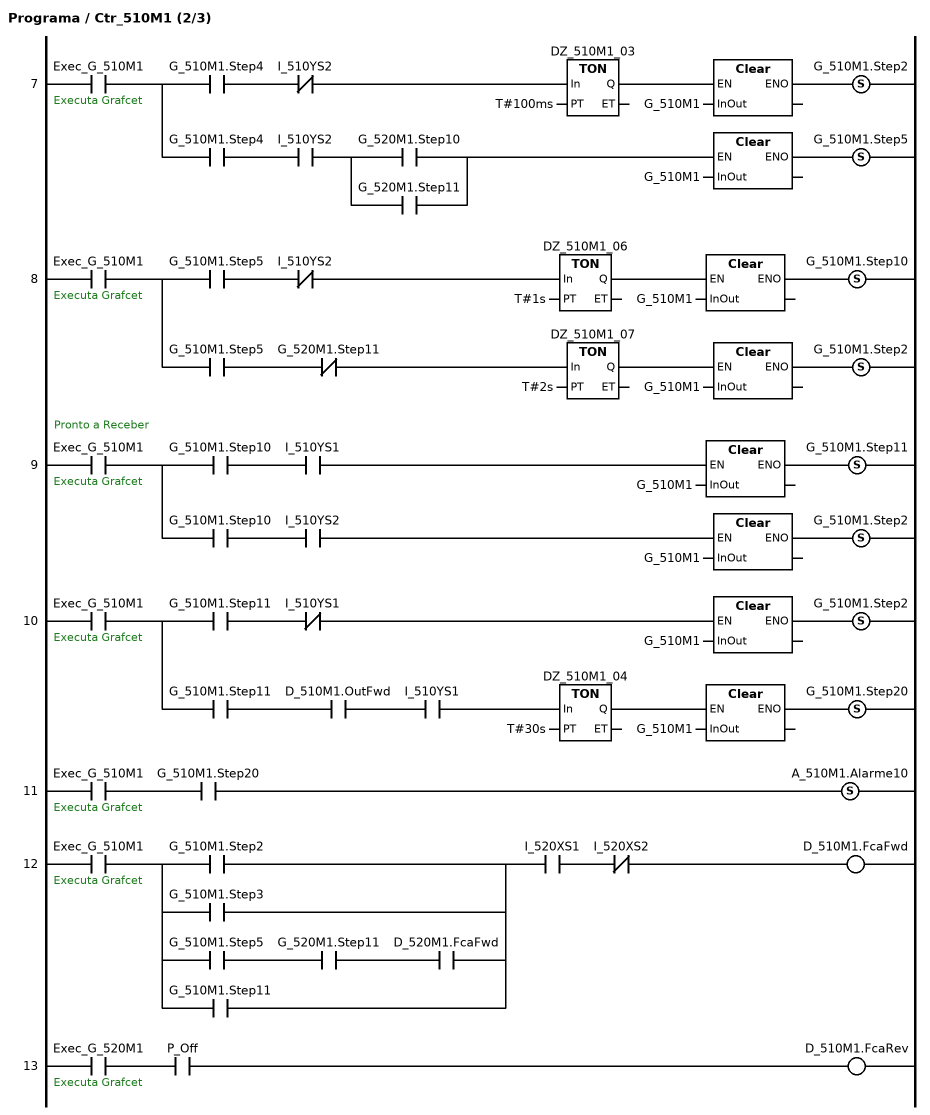
(* Rung 7 *)
DZ_510M1_03(In := Exec_G_510M1 AND G_510M1.Step4 AND NOT I_510YS2, PT := T#100ms);
IF DZ_510M1_03.Q THEN
    Clear(InOut := G_510M1);
    G_510M1.Step2 := TRUE;
END_IF;
_p211 := Exec_G_510M1 AND G_510M1.Step4 AND I_510YS2 AND (G_520M1.Step10 OR G_520M1.Step11);
IF _p211 THEN
    Clear(InOut := G_510M1);
    G_510M1.Step5 := TRUE;
END_IF;
(* Rung 8 *)
DZ_510M1_06(In := Exec_G_510M1 AND G_510M1.Step5 AND NOT I_510YS2, PT := T#1s);
IF DZ_510M1_06.Q THEN
    Clear(InOut := G_510M1);
    G_510M1.Step10 := TRUE;
END_IF;
DZ_510M1_07(In := Exec_G_510M1 AND G_510M1.Step5 AND NOT G_520M1.Step11, PT := T#2s);
IF DZ_510M1_07.Q THEN
    Clear(InOut := G_510M1);
    G_510M1.Step2 := TRUE;
END_IF;
(* Rung 9: Pronto a Receber *)
_p212 := Exec_G_510M1 AND G_510M1.Step10 AND I_510YS1;
IF _p212 THEN
    Clear(InOut := G_510M1);
    G_510M1.Step11 := TRUE;
END_IF;
_p213 := Exec_G_510M1 AND G_510M1.Step10 AND I_510YS2;
IF _p213 THEN
    Clear(InOut := G_510M1);
    G_510M1.Step2 := TRUE;
END_IF;
(* Rung 10 *)
_p214 := Exec_G_510M1 AND G_510M1.Step11 AND NOT I_510YS1;
IF _p214 THEN
    Clear(InOut := G_510M1);
    G_510M1.Step2 := TRUE;
END_IF;
DZ_510M1_04(In := Exec_G_510M1 AND G_510M1.Step11 AND D_510M1.OutFwd AND I_510YS1, PT := T#30s);
IF DZ_510M1_04.Q THEN
    Clear(InOut := G_510M1);
    G_510M1.Step20 := TRUE;
END_IF;
(* Rung 11 *)
IF Exec_G_510M1 AND G_510M1.Step20 THEN A_510M1.Alarme10 := TRUE; END_IF;
(* Rung 12 *)
D_510M1.FcaFwd := Exec_G_510M1 AND (G_510M1.Step2 OR G_510M1.Step3 OR (G_510M1.Step5 AND G_520M1.Step11 AND D_520M1.FcaFwd) OR G_510M1.Step11) AND I_520XS1 AND NOT I_520XS2;
(* Rung 13 *)
D_510M1.FcaRev := Exec_G_520M1 AND P_Off;

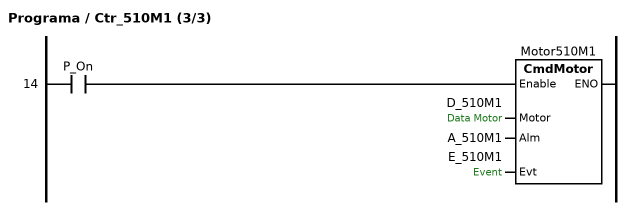
(* Rung 14 *)
Motor510M1(Enable := P_On, Motor := D_510M1, Alm := A_510M1, Evt := E_510M1);

(* Section Ctr_520M1: ladder, written here as Structured Text *)

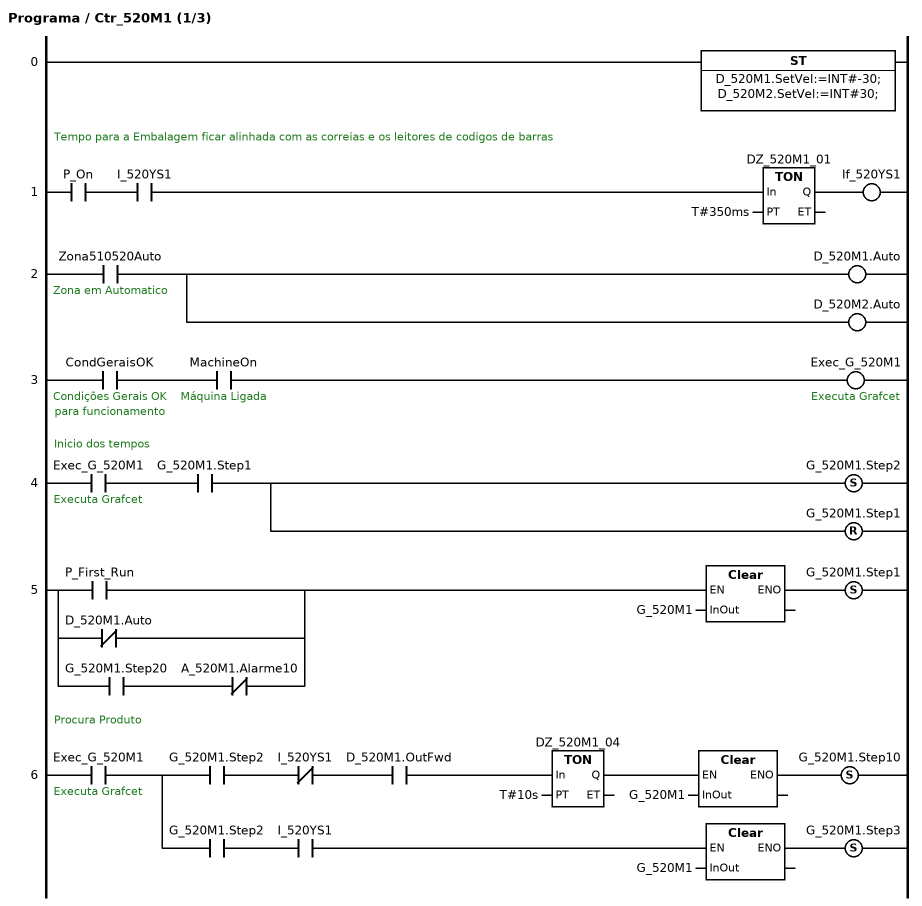
(* Rung 0 *)
D_520M1.SetVel:=INT#-30;
D_520M2.SetVel:=INT#30;
(* Rung 1: Tempo para a Embalagem ficar alinhada com as correias e os leitores de codigos de barras *)
DZ_520M1_01(In := P_On AND I_520YS1, PT := T#350ms);
If_520YS1 := DZ_520M1_01.Q;
(* Rung 2 *)
D_520M1.Auto := Zona510520Auto;
D_520M2.Auto := Zona510520Auto;
(* Rung 3 *)
Exec_G_520M1 := CondGeraisOK AND MachineOn;
(* Rung 4: Inicio dos tempos *)
_p215 := Exec_G_520M1 AND G_520M1.Step1;
IF _p215 THEN
    G_520M1.Step2 := TRUE;
    G_520M1.Step1 := FALSE;
END_IF;
(* Rung 5 *)
_p216 := P_First_Run OR NOT D_520M1.Auto OR (G_520M1.Step20 AND NOT A_520M1.Alarme10);
IF _p216 THEN
    Clear(InOut := G_520M1);
    G_520M1.Step1 := TRUE;
END_IF;
(* Rung 6: Procura Produto *)
DZ_520M1_04(In := Exec_G_520M1 AND G_520M1.Step2 AND NOT I_520YS1 AND D_520M1.OutFwd, PT := T#10s);
IF DZ_520M1_04.Q THEN
    Clear(InOut := G_520M1);
    G_520M1.Step10 := TRUE;
END_IF;
_p217 := Exec_G_520M1 AND G_520M1.Step2 AND I_520YS1;
IF _p217 THEN
    Clear(InOut := G_520M1);
    G_520M1.Step3 := TRUE;
END_IF;

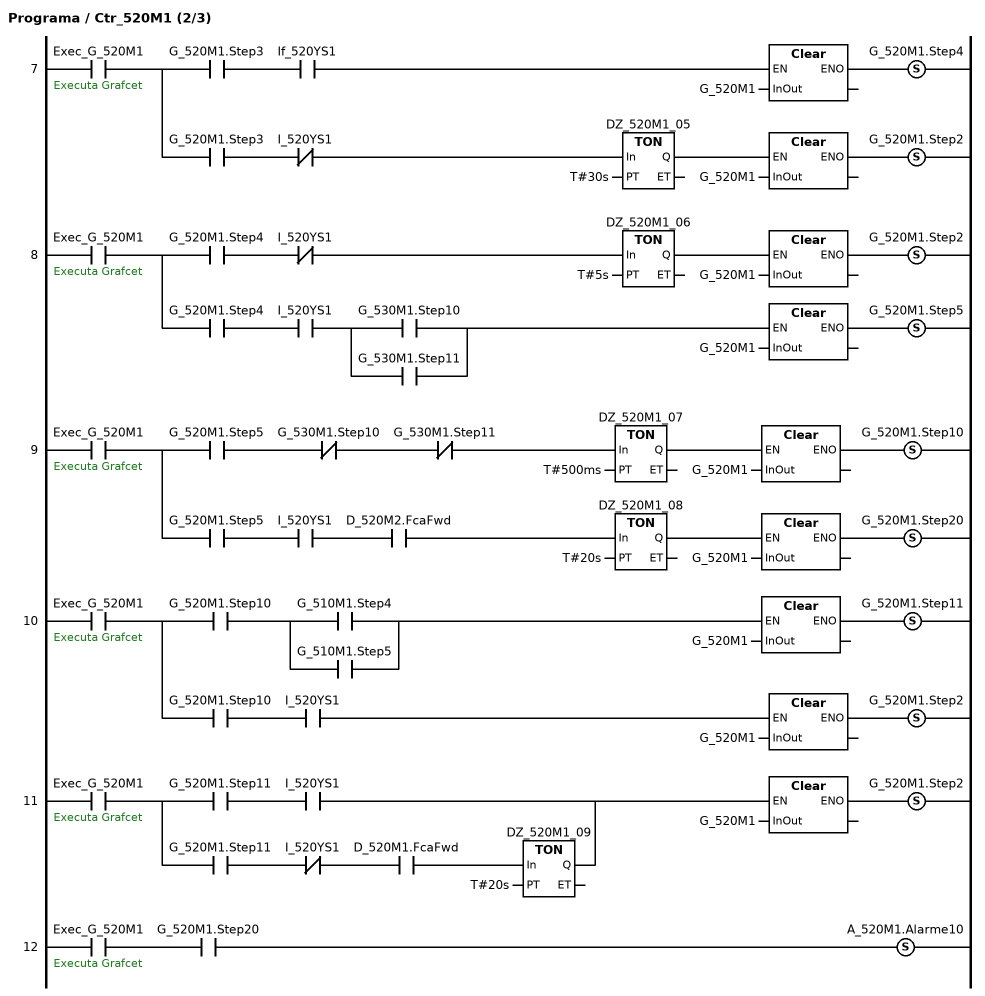
(* Rung 7 *)
_p218 := Exec_G_520M1 AND G_520M1.Step3 AND If_520YS1;
IF _p218 THEN
    Clear(InOut := G_520M1);
    G_520M1.Step4 := TRUE;
END_IF;
DZ_520M1_05(In := Exec_G_520M1 AND G_520M1.Step3 AND NOT I_520YS1, PT := T#30s);
IF DZ_520M1_05.Q THEN
    Clear(InOut := G_520M1);
    G_520M1.Step2 := TRUE;
END_IF;
(* Rung 8 *)
DZ_520M1_06(In := Exec_G_520M1 AND G_520M1.Step4 AND NOT I_520YS1, PT := T#5s);
IF DZ_520M1_06.Q THEN
    Clear(InOut := G_520M1);
    G_520M1.Step2 := TRUE;
END_IF;
_p219 := Exec_G_520M1 AND G_520M1.Step4 AND I_520YS1 AND (G_530M1.Step10 OR G_530M1.Step11);
IF _p219 THEN
    Clear(InOut := G_520M1);
    G_520M1.Step5 := TRUE;
END_IF;
(* Rung 9 *)
DZ_520M1_07(In := Exec_G_520M1 AND G_520M1.Step5 AND NOT G_530M1.Step10 AND NOT G_530M1.Step11, PT := T#500ms);
IF DZ_520M1_07.Q THEN
    Clear(InOut := G_520M1);
    G_520M1.Step10 := TRUE;
END_IF;
DZ_520M1_08(In := Exec_G_520M1 AND G_520M1.Step5 AND I_520YS1 AND D_520M2.FcaFwd, PT := T#20s);
IF DZ_520M1_08.Q THEN
    Clear(InOut := G_520M1);
    G_520M1.Step20 := TRUE;
END_IF;
(* Rung 10 *)
_p220 := Exec_G_520M1 AND G_520M1.Step10 AND (G_510M1.Step4 OR G_510M1.Step5);
IF _p220 THEN
    Clear(InOut := G_520M1);
    G_520M1.Step11 := TRUE;
END_IF;
_p221 := Exec_G_520M1 AND G_520M1.Step10 AND I_520YS1;
IF _p221 THEN
    Clear(InOut := G_520M1);
    G_520M1.Step2 := TRUE;
END_IF;
(* Rung 11 *)
DZ_520M1_09(In := Exec_G_520M1 AND G_520M1.Step11 AND NOT I_520YS1 AND D_520M1.FcaFwd, PT := T#20s);
_p222 := (Exec_G_520M1 AND G_520M1.Step11 AND I_520YS1) OR DZ_520M1_09.Q;
IF _p222 THEN
    Clear(InOut := G_520M1);
    G_520M1.Step2 := TRUE;
END_IF;
(* Rung 12 *)
IF Exec_G_520M1 AND G_520M1.Step20 THEN A_520M1.Alarme10 := TRUE; END_IF;

